FUNCTION Convert_REAL_TO_LREAL : Hresult
VAR_INPUT
	in : REAL;
	out : REFERENCE TO LREAL;
END_VAR

out := REAL_TO_LREAL(in);

END_FUNCTION

(* stored: Version 1.1.0.1, ProductVersion 3.1.4024.12
   POU Convert_REAL_TO_LREAL: Id {2cda2b08-9535-4a1f-84c0-80296f6667b5}, SpecialFunc None *)
